(* PLC project OOP_Curso, Beckhoff Automation GmbH TwinCAT PLC Control 3.5.13.21 *)
(* stored: creationDateTime 2023-03-18T11:24:11.1041748, modificationDateTime 2023-03-18T11:24:11.1090589 *)

PROGRAM _07_Herencia
VAR
	Padre: FB_Padre;
	Hijo : FB_Hijo;
	mot : Motor;
	pump: Pump;
	
	a:INT:=10;
	b:INT:=20;
	c,d,e,f,g,h,i:INT;
	
	vel:INT:=1;
	bOn : BOOL;
	bStatusxOnMotor : BOOL;
	bStatusxOnPump : BOOL;
END_VAR

            Padre(iIn1:=a);
padre.iPadreVar;
c:= padre.mDouble();
d:= padre.mMultiply();

//Se Heradan todos los Métodos y Atributos(Propiedades), también Hereda la SubClase (Hijo) las variables de la SuperClase (Padre).
hijo(iIn1:=a, iIn2:=b);
//el valor de la variable en el Hijo y en el Padre no son iguales, ya que lo que esta sucediendo dentro del area principal del Padre no se ejecuta en el Hijo...
//esto es debido a que el codigo del area principal no se herada del Padre al Hijo...
hijo.iPadreVar; 
e:= hijo.mDouble();
//se puede sobreescribir un metodo del Padre en el Hijo..., la Herencia posibilita la sobreescritura de los Metodos...
f:= hijo.mMultiply();
g:= hijo.mMinus(minus:=17);
h:= hijo.mSuperMultiply();

//Motor SuperClase
mot(iSpeed:= vel);
mot.iAngle;
IF bOn THEN
	mot.TurnON();
ELSE
	mot.TurnOff();
END_IF

bStatusxOnMotor:= mot.StatusxOn;

//Bomba SubClase de Motor
pump(iSpeed:= vel);
pump.iAngle;
IF bOn THEN
	pump.TurnON();
ELSE
	pump.TurnOff();
END_IF

bStatusxOnPump:= pump.StatusxOn;




          
END_PROGRAM

FUNCTION_BLOCK FB_Hijo EXTENDS FB_Padre
VAR_INPUT
	iIn2:int;
END_VAR
VAR_OUTPUT
END_VAR
VAR
END_VAR

            
          

METHOD mMinus : INT
VAR_INPUT
	minus:INT;
END_VAR
                  mMinus := iIn1 - minus;
                
END_METHOD

METHOD mMultiply : INT
VAR_INPUT
END_VAR
                  //Hemos Sobreescrito el metodo del Padre. (superclase).

mMultiply:= THIS^.iIn1 * iIn2;


                
END_METHOD

METHOD mSuperMultiply : INT
VAR_INPUT
END_VAR
                  //Accedemos al metodo del padre con SUPER^.

mSuperMultiply := 10 * SUPER^.mMultiply();




                
END_METHOD
END_FUNCTION_BLOCK

FUNCTION_BLOCK FB_Padre
VAR_INPUT
	iIn1: INT;
END_VAR
VAR_OUTPUT
	iOut:INT;
END_VAR
VAR
	iPadreVar:INT:= 42;
	iPadreTime: TON:=(in:=TRUE, pt:=T#1S);
END_VAR

            iPadreTime();
IF iPadreTime.Q THEN
	iPadreVar:= iPadreVar+iIn1;
	iPadreTime.IN:= FALSE;
ELSE
	iPadreTime.IN:= TRUE;
END_IF
          

METHOD mDouble : INT
VAR_INPUT
END_VAR
                  mDouble:= iIn1+iIn1;
                
END_METHOD

METHOD mMultiply : INT
VAR_INPUT
END_VAR
                  mMultiply := iIn1*5;
                
END_METHOD
END_FUNCTION_BLOCK

FUNCTION_BLOCK Motor
VAR_INPUT
	iSpeed :INT;
END_VAR
VAR_OUTPUT
	iOut:INT;
END_VAR
VAR
	iAngle:INT:=42;
	xOn: BOOL;
	iPapaTime: TON:=(in:=TRUE,pt:=t#1s);
END_VAR

            iPapaTime(in:=xOn, pt:=T#1S);
UpdateAngle();
          

METHOD TurnOff : BOOL
VAR_INPUT
END_VAR
                  xOn:= false;
                
END_METHOD

METHOD TurnON : BOOL
VAR_INPUT
END_VAR
                  xOn:= true;
                
END_METHOD

METHOD UpdateAngle : BOOL
VAR_INPUT
END_VAR
                  IF ipapatime.q THEN
	iangle:= iangle+ispeed;
	IF iangle>360 THEN
		iangle:=0;
	END_IF
	ipapatime.IN:= FALSE;
ELSE
	ipapatime.IN:= TRUE;
END_IF
                
END_METHOD

PROPERTY StatusxOn : BOOL
GET
VAR
END_VAR
                    StatusxOn:= xOn;
                  
END_GET
END_PROPERTY
END_FUNCTION_BLOCK

FUNCTION_BLOCK Pump EXTENDS Motor
VAR_INPUT
END_VAR
VAR_OUTPUT
END_VAR
VAR
END_VAR

            iPapaTime(in:=xOn, pt:=T#1S);
UpdateAngle();
          

METHOD UpdateAngle : BOOL
VAR_INPUT
END_VAR
                  IF ipapatime.q THEN
	//iangle:= iangle+ispeed;
	iangle:= iangle+ispeed*100;
//	IF iangle>360 THEN
//		iangle:=0;
//	END_IF
	ipapatime.IN:= FALSE;
ELSE
	ipapatime.IN:= TRUE;
END_IF
                
END_METHOD
END_FUNCTION_BLOCK
